{attribute 'linkalways'} 
{attribute 'no_explicit_call' := 'This FB is a CLASS and must be accessed using methods or properties'}
{attribute 'enable_dynamic_creation'}
FUNCTION_BLOCK Node_F_VN_PointToPointDirection_TcVnPoint2_DINT EXTENDS VisionNode
VAR
    aPoint1 : _TcVnPoint2_DINT;
    aPoint2 : _TcVnPoint2_DINT;
    aDirection : _TcVnVector2_LREAL;
    bNormalize : _BOOL(FALSE);
    hrPrev : _HRESULT(S_OK);
	hresult : _HRESULT(S_OK);
END_VAR

METHOD PUBLIC  Clone : I_Node
VAR
	pNode : POINTER TO Node_F_VN_PointToPointDirection_TcVnPoint2_DINT;
END_VAR
pNode := __NEW(Node_F_VN_PointToPointDirection_TcVnPoint2_DINT);
Clone := pNode^;
END_METHOD

METHOD FB_init : BOOL
VAR_INPUT
	bInitRetains : BOOL; // if TRUE, the retain variables are initialized (warm start / cold start)
	bInCopyCode : BOOL;  // if TRUE, the instance afterwards gets moved into the copy code (online change)
END_VAR
AddInput('aPoint1', aPoint1);
AddInput('aPoint2', aPoint2);
AddParameter('bNormalize', bNormalize);
AddInput('hrPrev', hrPrev);
AddOutput('aDirection', aDirection);
AddOutput('hresult',hresult);
END_METHOD

METHOD PROTECTED OnExecute
hresult.Value := F_VN_PointToPointDirection_TcVnPoint2_DINT(
    aPoint1 := aPoint1.Value,
    aPoint2 := aPoint2.Value,
    aDirection := aDirection.Value,
    bNormalize := bNormalize.Value,
	hrPrev:= hrPrev.Value);
END_METHOD

METHOD PUBLIC PreExecutionCheck
VAR_INPUT
	Check : I_PreExecutionChecks;
END_VAR
END_METHOD

END_FUNCTION_BLOCK

(* stored: Version 1.1.0.1, ProductVersion 3.1.4024.15
   POU Node_F_VN_PointToPointDirection_TcVnPoint2_DINT: Id {c7a85354-384f-078f-2094-8e85dd317d44}, SpecialFunc None
   Folder Constructor: Id {c6b97200-c93e-056d-1a5b-181bad3a6c39}
   Method Clone: Id {64b95ee2-b5c7-09a2-1e5a-b185b6cde42b}
   Method FB_init: Id {a22bdbda-0f51-0fe2-2ccc-d57da89c773d}
   Method OnExecute: Id {466c8932-05b7-0e8c-35e4-ac60a2c455d0}
   Method PreExecutionCheck: Id {586f98ea-d92f-0944-1fae-054914230b9b} *)
